FUNCTION_BLOCK FB_Combined
VAR_INPUT
    bEnabled : BOOL;
    nValue   : INT;
    rScale   : REAL;
    sLabel   : STRING;
END_VAR
VAR_OUTPUT
    nResult  : INT;
    rResult  : REAL;
    sStatus  : STRING;
END_VAR
VAR
    bActive  : BOOL;
END_VAR

bActive := bEnabled;
IF bActive THEN
    nResult := nValue;
    rResult := INT_TO_REAL(nValue) * rScale;
    sStatus := CONCAT(sLabel, ' enabled');
ELSE
    nResult := 0;
    rResult := 0.0;
    sStatus := CONCAT(sLabel, ' disabled');
END_IF;

PROPERTY Status : STRING
END_PROPERTY

METHOD Reset : BOOL
VAR_INPUT
END_VAR
END_METHOD

ACTION Apply:

END_ACTION

END_FUNCTION_BLOCK

(* stored: Version 1.1.0.1, ProductVersion 3.1.4024.10
   POU FB_Combined: KindOfPOU Element
   Method Reset: KindOfMethod Element
   Action Apply: KindOfAction Element *)
